{attribute 'GeneratedUsingTerminal: EL3051-0000-0017'}
{attribute addProperty BoxType "EL3051-0000-0017"}
{attribute addProperty Id "AI_StandardAT %I*AI_Standard_4A3944819WcStateAT %I*WcState_9091E0EB2InfoDataAT %I*InfoData_32EB74EA10"}
{attribute addProperty CRC "893334239"}
{attribute addProperty Size "21"}
TYPE EL3051_353F32DF :
STRUCT
	{attribute addProperty Name "AI_Standard"}
	AI_Standard : AI_Standard_4A394481;
	{attribute addProperty Name "WcState"}
	WcState : WcState_9091E0EB;
	{attribute addProperty Name "InfoData"}
	InfoData : InfoData_32EB74EA;
END_STRUCT
END_TYPE

(* stored: Version 1.2.0.0, ProductVersion 3.1.4024.9
   DUT EL3051_353F32DF: Id {18aa85c1-7690-4d77-87a2-88b0ba403b39} *)
